// TIA Portal V19 export
TYPE "typeDataToSafety"
// Information sent from the standard program to the safety program
// stored: Access Published, IsFailsafeCompliant true, Namespace Safety
   STRUCT
      ackSafetyFromHmi : Int;   // Acknowledge variable from operator control or monitoring system
      ackSafetyGlobal : Bool;   // Acknowledge command to ack all safety
      ackFromUnit : Bool;   // Acknowledge command comming from Unit
   END_STRUCT;
END_TYPE
